DEVICE_TYPE UAO_RT (* UAO Runtime running on a PC (Windows or Linux) *)
  (* Standard: 61499 ITA; Description: Copyright (c) 2017 Aimirim STI *)
  (* Version 1.0, 2024-04-01, Pedro Ricardo; Felipe Adriano, Aimirim STI, Initial version *)
  VAR_INPUT
    MGR_ID : WSTRING := "localhost:51499"; (* Device manager socket ID *)
    SSL : BOOL := FALSE; (* Use SSL encryption with the device *)
  END_VAR
END_DEVICE_TYPE
